{attribute 'qualified_only'}
VAR_GLOBAL CONSTANT
	//All robot values are in mm
	PICKUP_AREA_DEPTH : LREAL := 60.0 * 10;
	PICKUP_AREA_WIDTH : LREAL := 60.0 * 10;
	
	//Values in mm
	DISTANCE_TO_PICKUP_AREA : LREAL := 90.0;	//Real: 90mm
	ARM_BASE_HEIGHT : LREAL := 310;
	GRABBER_HEIGHT : LREAL := 0.0;
	ARM_1_LENGTH : LREAL := 340.0;
	ARM_2_LENGTH : LREAL := 265.0;
	ARM_3_LENGTH : LREAL := 170.0;
	Pi : LREAL := 3.141592653589793238463;
	
	DROPOFF_X : LREAL := 450.0;	//MM	//TODO: Use DEPTH/2
	DROPOFF_Z : LREAL := PICKUP_AREA_WIDTH / 2;	//MM
	//Height is taken from the pickedup target
	DROPOFF_BASE_OFFSET : LREAL := -90.0;	//Degrees
	

	
	//Values in degrees
	MAXIMUM_BASE_ROTATION_FROM_CENTER : LREAL := 120.0;
	
END_VAR

(* stored: Version 1.1.0.1, ProductVersion 3.1.4024.12
   GVL GVL_RobotArmConstants: Id {ef61bbec-f38a-46b1-ba77-40b840afe4d2} *)
